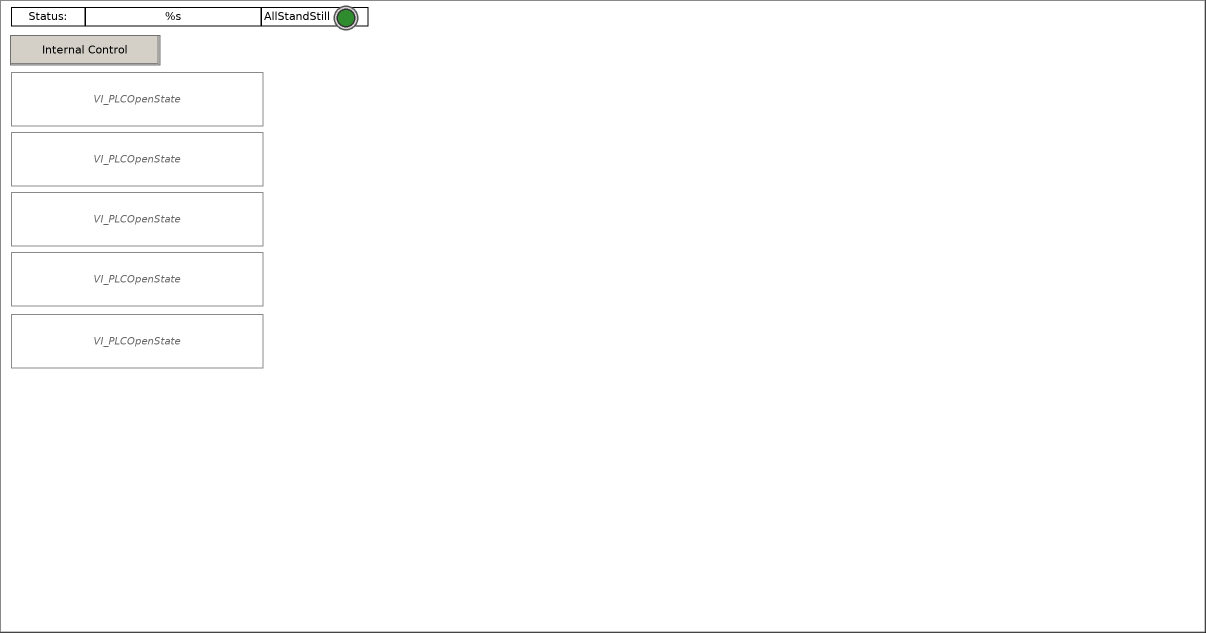
VISUALIZATION VI_GroupCAVisu  // 1206x633
VAR_IN_OUT
	gca : FB_GroupCA;
END_VAR
VAR
	stTableStruct : ARRAY [1..25] OF stTableStructx10;
END_VAR
    Rectangle (0,0 1206x633)
    Rectangle (85,7 176x19), "%s", text variable: gca.eGroupState, text list: 'GroupState_txt'
    Frame (11,72 252x54)
        shows VI_PLCOpenState(bExecute := gca.fbEnable.Execute, sName := 'Enable', bBusy := gca.fbEnable.Busy, bDone := gca.fbEnable.Done, bError := gca.fbEnable.Error, bCommandAborted := gca.bTmp, ErrorID := gca.fbEnable.ErrorId)
    Frame (11,132 252x54)
        shows VI_PLCOpenState(bExecute := gca.fbDisable.Execute, sName := 'Disable', bBusy := gca.fbDisable.Busy, bDone := gca.fbDisable.Done, bError := gca.fbDisable.Error, bCommandAborted := gca.bTmp, ErrorID := gca.fbDisable.ErrorId)
    Frame (11,192 252x54)
        shows VI_PLCOpenState(bExecute := gca.fbHalt.Execute, sName := 'Halt', bBusy := gca.fbHalt.Busy, bDone := gca.fbHalt.Done, bError := gca.fbHalt.Error, bCommandAborted := gca.fbHalt.CommandAborted, ErrorID := gca.fbHalt.ErrorId)
    Frame (11,252 252x54)
        shows VI_PLCOpenState(bExecute := gca.fbReset.Execute, sName := 'Reset', bBusy := gca.fbReset.Busy, bDone := gca.fbReset.Done, bError := gca.fbReset.Error, bCommandAborted := gca.bTmp, ErrorID := gca.fbReset.ErrorId)
    Rectangle (11,7 74x19), "Status:", text variable: gca.eGroupState
    Button (10,35 150x30), "Internal Control", tooltip "Enable Visu Control, all methods will be locked"
        toggle gca.bInternalControl
    Frame (11,314 252x54)
        shows VI_PLCOpenState(bExecute := gca.fbUnGroupAll.Execute, sName := 'UnGroupAll', bBusy := gca.fbUnGroupAll.Busy, bDone := gca.fbUnGroupAll.Done, bError := gca.fbUnGroupAll.Error, bCommandAborted := gca.bTmp, ErrorID := gca.fbUnGroupAll.ErrorId)
    Rectangle (261,7 107x19), "AllStandStill"
    Lamp1 (332,4 28x28), variable: gca.bAllStandStill, style: Lamp-Lamp1-Green
END_VISUALIZATION

(* stored: Version 1.1.0.1, ProductVersion 3.1.4024.11
   Visu VI_GroupCAVisu: Id {00677720-ca43-418c-8d95-dab0a9ceb448} *)
